// TIA Portal V18 export
// export: Created 2026-03-12T16:04:33.8104026Z, ExportSetting WithDefaults, DisplayName Totally Integrated Automation Portal, DisplayVersion V18 Update 5, DisplayName TIA Portal Openness, DisplayVersion V18 Update 5, DisplayName TIA Portal Version Control Interface, DisplayVersion V18, DisplayName SINAMICS Startdrive Advanced, DisplayVersion V18, DisplayName SINAMICS Startdrive G130, G150, S120, S150, SINAMICS MV, S210, DisplayVersion V18, DisplayName SINAMICS Startdrive G110M, G120, G120C, G120D, G120P, G115D, DisplayVersion V18, DisplayName STEP 7 Professional, DisplayVersion V18 Update 5, DisplayName STEP 7 Safety, DisplayVersion V18, DisplayName WinCC Professional, DisplayVersion V18 Update 5
FUNCTION_BLOCK "FB CONTADOR"   // FB7, LAD
TITLE = Function Block MINUTEIRO - Contador de Minutos
{ S7_Optimized_Access := 'TRUE' }
VERSION : 0.1
// Bloco para realizar a contagem de quantos minutos cada motor/bomba passou ligado.
// stored: AutoNumber true, IsIECCheckEnabled false, IsRetainMemResEnabled false, MemoryReserve 100, SetENOAutomatically false, UDAEnableTagReadback false
   VAR_INPUT
      INPUT_LIGADO : Bool;   // Entrada do sinal de falha instanciado na Network 1
      INPUT_RESET_MINUTEIRO : Bool;   // Entrada do sinal de reset minuteiro (minutos trabalhadas da bomba)
   END_VAR
   VAR_OUTPUT
      SEGUNDEIRO : UInt;   // Saída do segundeiro (segundos trabalhados da bomba)
      MINUTEIRO : Real;   // Saída do minuteiro (minutos trabalhados da bomba)
      HORIMETRO : Real;   // Saída do horimetro (horas trabalhados da bomba)
   END_VAR
   VAR
      RESET_SEGUNDO : Bool;   // Comando para zerar os minutos acumuladas
      MINUTO : Bool;   // Pulso para contador de minutos
      COUNT_MINUTO : Bool;   // Contador de minutos
      RESET_MINUTO : Bool;   // Reset do contador de minutos
      SEGUNDOS : UInt;   // Segundos armazenados
      TIMER_SEGUNDO : IEC_COUNTER;   // Bloco contador de segundos
   END_VAR
BEGIN

REGION Network 1: Comando para zerar os minutos acumuladas
   // TIMER_SEGUNDO: Bloco contador de segundos
   // TIMER_MINUTO: Bloco contador de minutos
   // INC: Incremento de horas
   // RESET_MINUTEIRO: Comando para zerar os minutos acumulados
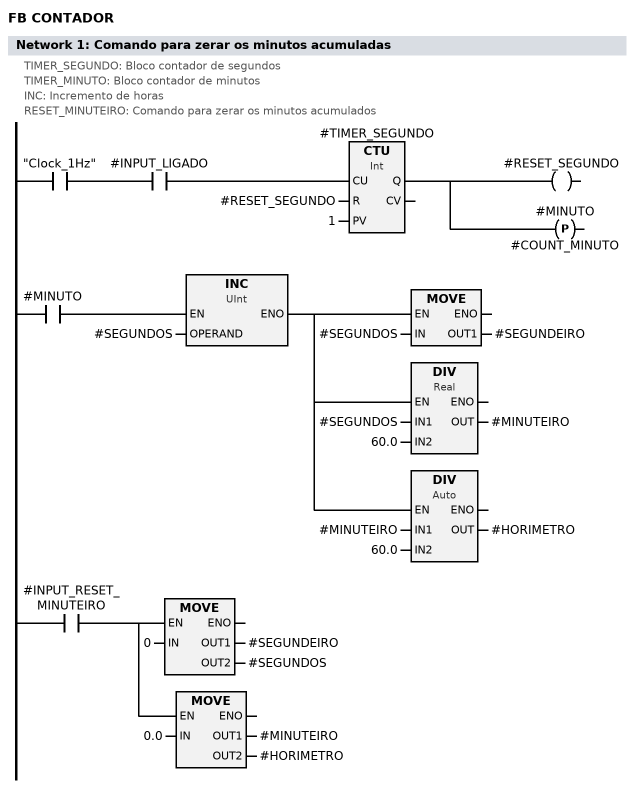
   #TIMER_SEGUNDO.CTU(CU := "Clock_1Hz" AND #INPUT_LIGADO, R := #RESET_SEGUNDO, PV := 1);
   #RESET_SEGUNDO := #TIMER_SEGUNDO.Q;
   #MINUTO := #TIMER_SEGUNDO.Q AND NOT #COUNT_MINUTO;   // rising edge
   #COUNT_MINUTO := #TIMER_SEGUNDO.Q;
   IF #MINUTO THEN
       #SEGUNDOS := #SEGUNDOS + 1;
       #SEGUNDEIRO := #SEGUNDOS;
       #MINUTEIRO := #SEGUNDOS / 60.0;
       #HORIMETRO := #MINUTEIRO / 60.0;
   END_IF;
   IF #INPUT_RESET_MINUTEIRO THEN
       #SEGUNDEIRO := 0;
       #SEGUNDOS := 0;
       #MINUTEIRO := 0.0;
       #HORIMETRO := 0.0;
   END_IF;
END_REGION
END_FUNCTION_BLOCK
